// TwinCAT 3 PLC project PLC2_Client
// ProgramVersion: 3.1.4024.0
// libraries:
//   Tc2_DataExchange, * (Beckhoff Automation GmbH)
//   Tc2_Standard, * (Beckhoff Automation GmbH)
//   Tc2_System, * (Beckhoff Automation GmbH)
//   Tc3_Module, * (Beckhoff Automation GmbH)
// project tree:
//   / PlcTask.TcTTO
//   POUs/ P_Client.TcPOU
// (motion and I/O tree: see PLC project plc1_server)
// real-time tasks:
//   TASK PlcTask: cycle T#10ms, priority 20, ADS port 350
//   TASK PlcTask1: cycle T#10ms, priority 21, ADS port 351

CONFIGURATION PLC2_Client
    RESOURCE PLC ON TwinCAT3
        TASK PlcTask(INTERVAL := T#10ms, PRIORITY := 21);
        PROGRAM P_Client WITH PlcTask : P_Client;
    END_RESOURCE
END_CONFIGURATION

// ---- POUs/P_Client.TcPOU
PROGRAM P_Client
VAR
	//odczyt po adresie
	fbRead_Address			: ADSREAD;  
	sVarRead_Address		: STRING;					// zmienna przechowująca odczytane dane 
	bRead1					: BOOL;
	//zapis po adresie 
	fbWrite_Address			: ADSWRITE;
	sVarWrite_Address		: STRING:='Automation'; 	//zmienna przechowująca dane do wysłania 
	bWrite1					: BOOL;
	//odczyt po nazwie
	fbRead_Symbol			: FB_ReadAdsSymByName;
	bRead2					: BOOL;
	sVarRead_Symbol			: STRING;					// zmienna przechowująca odczytane dane 
	//zapis po nazwie 
	fbWrite_Symbol			: FB_WriteAdsSymByName;
	sVarWrite_Symbol		: STRING:='EtherCAT'; 		// zmienna przechowująca dane do wysłania 
	bWrite2					: BOOL;
END_VAR

fbRead_Address(
	NETID:='' , 
	PORT:=851 , 
	IDXGRP:=16#4020 , 	// 16#4020 odnosi się do adresacji %MB
	IDXOFFS:=0 , 		// offset wynika z adresu, np. %MB0 --> offset 0
	LEN:=SIZEOF(sVarRead_Address) , 
	DESTADDR:=ADR(sVarRead_Address) , 
	READ:=bRead1 , 
	TMOUT:= , 
	BUSY=> , 
	ERR=> , 
	ERRID=> );
	
fbWrite_Address(
	NETID:='' , 
	PORT:=851 , 
	IDXGRP:=16#4020 , // 16#4020 odnosi się do adresacji %MB
	IDXOFFS:=100 ,    // offset wynika z adresu, np. %MB100 --> offset 100
	LEN:=SIZEOF(sVarWrite_Address) , 
	SRCADDR:=ADR(sVarWrite_Address) , 
	WRITE:=bWrite1 , 
	TMOUT:= , 
	BUSY=> , 
	ERR=> , 
	ERRID=> );
	
fbRead_Symbol(
	bRead:=bRead2 , 
	sNetId:='' , 
	nPort:=851 , 
	sVarName:='P_Server.sVar2_Read' , 
	nDestAddr:=ADR(sVarRead_Symbol) , 
	nLen:=SIZEOF(sVarRead_Symbol) , 
	tTimeout:= , 
	eComMode:= , 
	bClearOnError:= , 
	bBusy=> , 
	bError=> , 
	nErrorId=> );
	
fbWrite_Symbol(
	bWrite:=bWrite2 , 
	sNetId:='' , 
	nPort:=851 , 
	sVarName:='P_Server.sVar2_Write' , 
	nSrcAddr:= ADR(sVarWrite_Symbol), 
	nLen:=SIZEOF(sVarWrite_Symbol) , 
	tTimeout:= , 
	eComMode:= , 
	bBusy=> , 
	bError=> , 
	nErrorId=> );

END_PROGRAM
